FUNCTION F_softsign : lreal
VAR_INPUT
	x : LREAL;
END_VAR

F_softsign := x / (abs(x) + 1);

END_FUNCTION

(* stored: Version 1.1.0.1, ProductVersion 3.1.4024.12
   POU F_softsign: Id {8b3be192-4fc8-4ea0-b942-0ae23a6c8559}, SpecialFunc None *)
